// LS Electric XG5000 project: 8_20_mini_project
// PLC LSPLC

PROGRAM NewProgram (task: 스캔 프로그램)

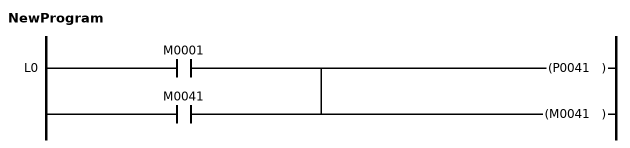
; L0
LOAD      M0001
OR        M0041
OUT       P0041
OUT       M0041